(* LS Electric XG5000 project: 241007_펑션블록CTU *)
(* PLC LSPLC *)
(* module base 0 slot 0: 입력 모듈:XGI-D22A/B (DC 24V 입력, 16점 (전류소스 싱크공용/ 전류소스 입력)) *)
(* module base 0 slot 1: 출력 모듈:XGQ-RY1A (릴레이 출력, 8점 (2A용, 단독 COM.)) *)

PROGRAM NewProgram (* task: 스캔 프로그램 *)
VAR
    C1 : CTU_INT;
    C2 : CTD_INT;
    램프1 AT %QX0.1.0 : BOOL;
    램프2 AT %QX0.1.1 : BOOL;
    리셋 AT %IX0.0.3 : BOOL;
    시작1 AT %IX0.0.0 : BOOL;
    시작2 AT %IX0.0.2 : BOOL;
END_VAR

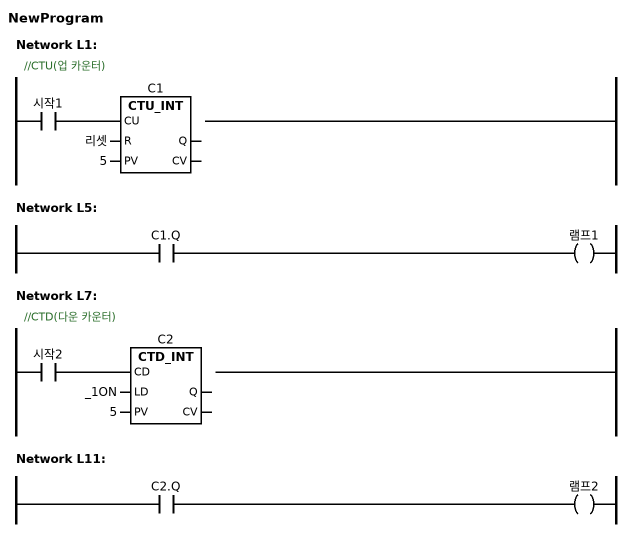
(* //CTU(업 카운터) *)
(* Rung L1 *)
C1(CU := 시작1, R := 리셋, PV := 5);
(* Rung L5 *)
램프1 := C1.Q;
(* //CTD(다운 카운터) *)
(* Rung L7 *)
C2(CD := 시작2, LD := _1ON, PV := 5);
(* Rung L11 *)
램프2 := C2.Q;
END_PROGRAM